TYPE stHMI_ROB_AXIS :
STRUCT
    ConfigurationValid : BOOL;
    AtMinLimit : BOOL;
    AtMaxLimit : BOOL;
    InPosition : BOOL;
END_STRUCT
END_TYPE

(* stored: Version 1.1.0.1, ProductVersion 3.1.4026.18
   DUT stHMI_ROB_AXIS: Id {1b002753-a75e-4568-a17d-b12d3acf058e} *)
